    !*********************************************************
    ! Routine:  PrensaCtrlColoc()
    !*********************************************************
    FUNC bool PrensaCtrlColoc()
        VAR bool bPrnColocKo:=FALSE;

        IF DI_P240_PrnAuto=1 THEN
            USR_MsgWaitDI DI_P242_PrnOkColoc,s_AttesaDepoPrensa{nIdioma};
            WaitDI DI_P242_PrnOkColoc,1\MaxTime:=nTempoMaxDIPrnColoc\TimeFlag:=bPrnColocKo;
            IF bPrnColocKo=TRUE THEN
                Set DO_V08_LuzVermelha;
                ROB_AlarmeAcustico(2);
                USR_Print(s_CaricoPrensaKo{nIdioma});
                WaitTime nTempoMensAnom;
                Reset DO_V08_LuzVermelha;
                RETURN FALSE;
            ELSE
                RETURN TRUE;
            ENDIF
        ELSE
            Set DO_V08_LuzVermelha;
            ROB_AlarmeAcustico(2);
            USR_Print(s_AutomaticoPrensa{nIdioma});
            WaitTime nTempoMensAnom;
            Reset DO_V08_LuzVermelha;
            RETURN FALSE;
        ENDIF

    ENDFUNC

    !*********************************************************
    ! Routine:  PrensaCtrlPega()
    !*********************************************************
    FUNC bool PrensaCtrlPega()
        VAR bool bPrnPegalKo:=FALSE;

        IF DI_P240_PrnAuto=1 THEN
            USR_MsgWaitDI DI_P243_PrnOkPega,s_AttesaPrelievoPrensa{nIdioma};
            WaitDI DI_P243_PrnOkPega,1\MaxTime:=nTempoMaxDIPrnPega\TimeFlag:=bPrnPegalKo;
            IF bPrnPegalKo=TRUE THEN
                Set DO_V08_LuzVermelha;
                ROB_AlarmeAcustico(2);
                USR_Print(s_ErrPrelievoPrensa{nIdioma});
                WaitTime nTempoMensAnom;
                Reset DO_V08_LuzVermelha;
                RETURN FALSE;
            ELSE
                RETURN TRUE;
            ENDIF
        ELSE
            Set DO_V08_LuzVermelha;
            ROB_AlarmeAcustico(2);
            USR_Print(s_AutomaticoPrensa{nIdioma});
            WaitTime nTempoMensAnom;
            Reset DO_V08_LuzVermelha;
            RETURN FALSE;
        ENDIF

    ENDFUNC

    !*********************************************************
    ! Routine:  mENF_Cuba()
    !*********************************************************
    PROC mENF_Cuba()

        USR_Print(s_CicloRaffr{nIdioma});

        !MoveJ ENF_p01, vmax, z100, USR_toolGarra\WObj:=wobjMDF;
        !MoveJ ENF_p02, vmax, z100, USR_toolGarra\WObj:=wobjMDF;
        !MoveJ ENF_p03, vmax, z50, USR_toolGarra\WObj:=wobjMDF;
        !MoveJ ENF_p04, vmax, z50, USR_toolGarra\WObj:=wobjMDF;

        ! ===>>> POSICAO de Esfriamento <<<===
        !MoveL ENF_pCuba, v800, fine, USR_toolGarra\WObj:=wobjMDF;
        MoveJ ENF_pCuba,v150,fine,USR_toolGarra\WObj:=wobjMDF;
        ! ======================================
        USR_Print(s_AttesaRaff{nIdioma});
        WaitTime nTempoEsfriam;

        MoveL ENF_p01,v150,z50,USR_toolGarra\WObj:=wobjMDF;
        MoveJ ENF_p11,v150,z50,USR_toolGarra\WObj:=wobjMDF;
        ! MoveJ ENF_p12, v100, z50, USR_toolGarra\WObj:=wobjMDF;

        ! ===> POSICAO de GOTEJAMENTO <===
        MoveL ENF_p20,v80,fine,USR_toolGarra\WObj:=wobjMDF;
        MoveL ENF_p30,v80,fine,USR_toolGarra\WObj:=wobjMDF;
        ! =================================
        USR_Print(s_AttesaSgocc{nIdioma});
        WaitTime nTempoGotejamento;

        MoveJ ENF_p22,v600,z100,USR_toolGarra\WObj:=wobjMDF;
        !MoveJ ENF_p23, v600, z100, USR_toolGarra\WObj:=wobjMDF;

    ENDPROC

    !*********************************************************
    ! Routine:  mDEP_UtilIntColoc()
    !*********************************************************
    PROC mDEP_UtilIntColoc()

        USR_Print(s_UtilDepo{nIdioma});

        MoveJ UTL_p01,v2000,z100,USR_toolGarra\WObj:=wobjMDF;
        !MoveJ UTL_p02, v2000, z100, USR_toolGarra\WObj:=wobjMDF;
        !MoveJ UTL_p03, v2000, z100, USR_toolGarra\WObj:=wobjMDF;
        !MoveL UTL_p04, v2000, z50, USR_toolGarra\WObj:=wobjMDF;
        MoveL Offs(UTL_pColoc,0,0,400),v600,fine,USR_toolGarra\WObj:=wobjMDF;

        ! ===>>> POSICAO DE COLOCACAO <<<===
        MoveL UTL_pColoc,v30,fine,USR_toolGarra\WObj:=wobjMDF;
        ! =====================================
        ROB_GarraAbrir;
        nTipoPcNaPinca:=0;
        bPcColocada:=TRUE;

        MoveL Offs(UTL_pColoc,0,0,200),v800,fine,USR_toolGarra\WObj:=wobjMDF;
        MoveJ UTL_p11,vmax,z100,USR_toolGarra\WObj:=wobjMDF;
        !MoveJ UTL_p12, v1500, z100, USR_toolGarra\WObj:=wobjMDF;

        ! control sensor
        IF (bHbltcSnsUtilInt=TRUE AND DI_W17_SnsUtilIntermedio=0) THEN
            USR_Print(s_UtilSnsDeact{nIdioma});
            Set DO_V08_LuzVermelha;
            ROB_AlarmeAcustico(2);
            Reset DO_P006_AnomaliaRobo;
            PulseDO\PLength:=2,DO_P006_AnomaliaRobo;
            USR_Print(s_AttesaReset{nIdioma});
            WaitDI DI_V01_ResetAllRob,1;
            Reset DO_V08_LuzVermelha;
        ENDIF

    ENDPROC

    !*********************************************************
    ! Routine:  mDEP_UtilIntRecoc()
    !*********************************************************
    PROC mDEP_UtilIntPega()

        USR_Print(s_UtilPrel{nIdioma});

        MoveJ UTL_p51,v5000,z100,USR_toolGarra\WObj:=wobjMDF;
        !MoveJ UTL_p52, vmax, z100, USR_toolGarra\WObj:=wobjMDF;
        !MoveJ UTL_p53, vmax, z100, USR_toolGarra\WObj:=wobjMDF;
        !MoveL UTL_p54, v1500, z50, USR_toolGarra\WObj:=wobjMDF;
        MoveL Offs(UTL_pPega,0,0,200),v800,fine,USR_toolGarra\WObj:=wobjMDF;

        ! ===>>> POSICAO DE RETIRADA <<<===
        MoveL UTL_pPega,v100,fine,USR_toolGarra\WObj:=wobjMDF;
        ! ==================================
        ROB_GarraFechar;
        nTipoPcNaPinca:=1;
        bPcColocada:=FALSE;

        MoveL Offs(UTL_pPega,0,0,200),v1000,fine,USR_toolGarra\WObj:=wobjMDF;
        !MoveJ UTL_p61, vmax, z100, USR_toolGarra\WObj:=wobjMDF;
        MoveJ UTL_p62,v1500,z100,USR_toolGarra\WObj:=wobjMDF;
        MoveJ UTL_p82,v1500,z100,USR_toolGarra\WObj:=wobjMDF;
        !MoveJ UTL_p72, vmax, z100, USR_toolGarra\WObj:=wobjMDF;

        ! control sensor
        IF (bHbltcSnsUtilInt=TRUE AND DI_W17_SnsUtilIntermedio=1) THEN
            USR_Print(s_UtilSnsAct{nIdioma});
            Set DO_W02_LuzAmarelo;
            ROB_AlarmeAcustico(2);
            Reset DO_P006_AnomaliaRobo;
            PulseDO\PLength:=2,DO_P006_AnomaliaRobo;
            WaitTime nTempoMensAnom;
            Reset DO_W02_LuzAmarelo;
        ENDIF

    ENDPROC

    !*********************************************************
    ! Routine:  mDEP_PrnColoc()
    !*********************************************************
    PROC mDEP_PrnColoc()

        USR_Print(s_DepositoPrensa{nIdioma});

        MoveJ PRN_p01,v2500,z100,USR_toolGarra\WObj:=wobjMDF;
        !
        ! Quebra de Rebarba...
        MoveJ pQuebraRebarba_00,v1500,z30,USR_toolGarra\WObj:=wobjMDF;
        MoveJ pQuebraRebarba_01,v800,z30,USR_toolGarra\WObj:=wobjMDF;
        MoveJ pQuebraRebarba_02,v600,z30,USR_toolGarra\WObj:=wobjMDF;
        MoveJ pQuebraRebarba_02,v1000,z30,USR_toolGarra\WObj:=wobjMDF;
        MoveJ pQuebraRebarba_00,v1500,z30,USR_toolGarra\WObj:=wobjMDF;
        !
        MoveJ PRN_p01,v2500,z100,USR_toolGarra\WObj:=wobjMDF;

        ! ===>>> POSICAO FUERA de la PRENSA!!! <<<===
        MoveJDO PRN_p02,v800,z100,USR_toolGarra\WObj:=wobjMDF,DO_V06_PrensaForaAreaTrab_User,0;
        ! ============================================

        MoveJ PRN_p03,v1000,z100,USR_toolGarra\WObj:=wobjMDF;
        !MoveL PRN_p04, v1000, z100, USR_toolGarra\WObj:=wobjMDF;
        !MoveJ PRN_p05, v800, z50, USR_toolGarra\WObj:=wobjMDF;
        !
        !    Defino a posicao de deposito como sendo uma para cada retirada da gaveta
        !
        TEST nRetirouDaGaveta
            CASE 1:
                PRN_pColoc := pDepositaPrensa_1;
            CASE 2:
                PRN_pColoc := pDepositaPrensa_2;
            CASE 3:
                PRN_pColoc := pDepositaPrensa_3;
            CASE 4:
                PRN_pColoc := pDepositaPrensa_4;
            CASE 5:
                PRN_pColoc := pDepositaPrensa_5;
            CASE 6:
                PRN_pColoc := pDepositaPrensa_6;
            DEFAULT:
                PRN_pColoc := PRN_pColoc;
                Stop;
        ENDTEST


        !
        !
        !pDepositaPrensa_1 := PRN_pColoc;
        !
        MoveJ Offs(PRN_pColoc,0,0,250),v400,fine,USR_toolGarra\WObj:=wobjMDF;

        ! ===>>> POSICAO de COLOCACAO <<<===
        MoveL PRN_pColoc,v200,fine,USR_toolGarra\WObj:=wobjMDF;
        ! ====================================

        ROB_GarraAbrir;
        nTipoPcNaPinca:=0;
        bPcColocada:=TRUE;

        !MoveL PRN_p10, v500, z10, USR_toolGarra\WObj:=wobjMDF;
        MoveL Offs(PRN_pColoc,0,0,200),v600,fine,USR_toolGarra\WObj:=wobjMDF;
        MoveL PRN_p11,v1000,z50,USR_toolGarra\WObj:=wobjMDF;
        !MoveJ PRN_p12, vmax, z100, USR_toolGarra\WObj:=wobjMDF;

        ! ===>>> POSICAO FUERA de la PRENSA!!! <<<===
        MoveJDO PRN_p13,v800,z5,USR_toolGarra\WObj:=wobjMDF,DO_V06_PrensaForaAreaTrab_User,1;
        ! ============================================

        MoveJ PRN_p14,vmax,fine,USR_toolGarra\WObj:=wobjMDF;

        USR_Print(s_StartPrensa{nIdioma});
        WaitTime\inpos,0;
        Reset DO_P242_PrnStartAposColoc;
        PulseDO\PLength:=1,DO_P242_PrnStartAposColoc;

        Reset DO_P033_PcColocPrensa;
        PulseDO\PLength:=1,DO_P033_PcColocPrensa;

        WaitDI DI_P242_PrnOkColoc,0\MaxTime:=1\TimeFlag:=bPrnErrStart1;
        IF bPrnErrStart1=TRUE THEN
            ROB_AlarmeAcustico(2);
            USR_Print(s_PrensaNonPartita{nIdioma});
            WaitTime nTempoMensAnom;
        ENDIF

    ENDPROC

    !*********************************************************
    ! Routine:  mDEP_PrnPega()
    !*********************************************************
    PROC mDEP_PrnPega()

        USR_Print(s_PrelievoPrensa{nIdioma});
        Set DO_W09_AbrirGarra;
        nTipoPcNaPinca:=0;
        bPcColocada:=TRUE;

        MoveJ PRN_p50,vmax,z100,USR_toolGarra\WObj:=wobjMDF;

        ! ===>>> POSICAO FUERA de la PRENSA!!! <<<===
        MoveJDO PRN_p51,vmax,z50,USR_toolGarra\WObj:=wobjMDF,DO_V06_PrensaForaAreaTrab_User,0;
        ! ============================================

        MoveJ PRN_p52,vmax,z100,USR_toolGarra\WObj:=wobjMDF;
        MoveJ PRN_p53,vmax,z100,USR_toolGarra\WObj:=wobjMDF;
        MoveL PRN_p54,vmax,z10,USR_toolGarra\WObj:=wobjMDF;

        ! ===>>> POSICAO de RETIRADA <<<===
        MoveL PRN_pPega,v300,fine,USR_toolGarra\WObj:=wobjMDF;
        ! ==================================

        IF bHbltcPrnPegaSoft=TRUE THEN
            SoftAct 1,100;
            ! SoftAct 2,10;
            ! SoftAct 3,10;
            SoftAct 4,10;
            SoftAct 5,10;
            SoftAct 6,10;
            WaitTime nTempoGarraFechar;
            !Tempo espera pasaje hacia ejes soft
        ENDIF

        ROB_GarraFechar;
        nTipoPcNaPinca:=1;
        bPcColocada:=FALSE;

        IF bHbltcPrnPegaSoft=TRUE THEN
            WaitTime 1;
            WaitTime\inpos,0;
            PRN_pTemp:=CRobT(\Tool:=USR_toolGarra\WObj:=wobjMDF);
            SoftDeact;
            MoveL Offs(PRN_pTemp,0,0,300),v100,fine,USR_toolGarra\WObj:=wobjMDF;
            WaitTime\inpos,0;
            SoftDeact;
        ENDIF

        MoveL PRN_p60,v1500,fine,USR_toolGarra\WObj:=wobjMDF;
        MoveL PRN_p61,vmax,fine,USR_toolGarra\WObj:=wobjMDF;
        MoveL PRN_p62,vmax,z100,USR_toolGarra\WObj:=wobjMDF;

        ! ===>>> POSICAO FUERA de la PRENSA!!! <<<===
        MoveJDO PRN_p63,vmax,z5,USR_toolGarra\WObj:=wobjMDF,DO_V06_PrensaForaAreaTrab_User,1;
        ! ============================================

        MoveJ PRN_p64,vmax,z100,USR_toolGarra\WObj:=wobjMDF;

        USR_Print(s_StartPrensa{nIdioma});
        WaitTime\inpos,0;
        Reset DO_P243_PrnStartAposPega;
        PulseDO\PLength:=1,DO_P243_PrnStartAposPega;

        Reset DO_P044_PcPegaPrensa;
        PulseDO\PLength:=1,DO_P044_PcPegaPrensa;

        WaitDI DI_P243_PrnOkPega,0\MaxTime:=1\TimeFlag:=bPrnErrStart2;
        IF bPrnErrStart2=TRUE THEN
            ROB_AlarmeAcustico(2);
            USR_Print(s_PrensaNonPartita{nIdioma});
            WaitTime nTempoMensAnom;
        ENDIF

    ENDPROC

    PROC PresaSoft()

        ROB_GarraAbrir;
        MoveL p01,v500,fine,USR_toolGarra\WObj:=wobjMDF;
        MoveL p02,v300,fine,USR_toolGarra\WObj:=wobjMDF;

        SoftAct 1,100;
        ! SoftAct 2,10;
        ! SoftAct 3,10;
        SoftAct 4,10;
        SoftAct 5,10;
        SoftAct 6,10;
        WaitTime nTempoGarraFechar;

        ROB_GarraFechar;

        WaitTime 1;
        WaitTime\inpos,0;
        pTemp:=CRobT(\Tool:=USR_toolGarra\WObj:=wobjMDF);
        MoveL Offs(pTemp,0,0,200),v300,fine,USR_toolGarra\WObj:=wobjMDF;
        WaitTime\inpos,0;
        SoftDeact;

        MoveL p01,v500,fine,USR_toolGarra\WObj:=wobjMDF;

    ENDPROC

    !*********************************************************
    ! Routine:  mDEP_PcPrensadaColoc()
    !*********************************************************
    PROC mDEP_PcPrensadaColoc()

        USR_Print(s_DepositoPrensati{nIdioma});

        MoveJ PRD_p01,vmax,z100,USR_toolGarra\WObj:=wobjMDF;
        MoveJ PRD_p02,vmax,z100,USR_toolGarra\WObj:=wobjMDF;
        MoveJ PRD_p03,vmax,z100,USR_toolGarra\WObj:=wobjMDF;
        MoveJ PRD_p04,v600,z20,USR_toolGarra\WObj:=wobjMDF;
        MoveL PRD_p05,v400,fine,USR_toolGarra\WObj:=wobjMDF;

        ! ===>>> POSICAO de COLOCACAO <<<===
        MoveL PRD_pColoc,v300,fine,USR_toolGarra\WObj:=wobjMDF;
        ! ====================================

        ROB_GarraAbrir;
        MoveL Offs(PRD_pColoc,0,0,120),v300,fine,USR_toolGarra\WObj:=wobjMDF;
        nTipoPcNaPinca:=0;
        bPcColocada:=TRUE;

        MoveL PRD_p10,v500,z50,USR_toolGarra\WObj:=wobjMDF;
        MoveL PRD_p11,vmax,z100,USR_toolGarra\WObj:=wobjMDF;
        MoveJ PRD_p12,vmax,z100,USR_toolGarra\WObj:=wobjMDF;
        MoveJ PRD_p13,vmax,z100,USR_toolGarra\WObj:=wobjMDF;
        MoveJ PRD_p14,vmax,z100,USR_toolGarra\WObj:=wobjMDF;

        Reset DO_P035_PcColocEsteiraRejeicao;
        PulseDO\PLength:=nTempPulsoEsteira,DO_P034_PcColocEsteiraBoa;

    ENDPROC

    !*********************************************************
    ! Routine:  mDEP_PcBoaColoc()
    !*********************************************************
    PROC mDEP_PcBoaColoc()

        IF bQualidade=TRUE THEN
            ROB_AlarmeAcustico(2);
            USR_Print(s_DepQualita{nIdioma});
        ELSE
            USR_Print(s_DepositoBuono{nIdioma});
        ENDIF

        MoveJ BUE_p01,vmax,z100,USR_toolGarra\WObj:=wobjMDF;
        MoveJ BUE_p02,vmax,z100,USR_toolGarra\WObj:=wobjMDF;
        MoveJ BUE_p03,vmax,z100,USR_toolGarra\WObj:=wobjMDF;
        MoveL BUE_p04,vmax,z100,USR_toolGarra\WObj:=wobjMDF;
        MoveL BUE_p05,v800,z50,USR_toolGarra\WObj:=wobjMDF;

        ! ===>>> POSICAO de COLOCACAO <<<===
        MoveL BUE_pColoc,v500,fine,USR_toolGarra\WObj:=wobjMDF;
        ! ====================================

        ROB_GarraAbrir;
        nTipoPcNaPinca:=0;
        bPcColocada:=TRUE;
        IF bQualidade=TRUE THEN
            bQualidade:=FALSE;
            Reset DO_W02_LuzAmarelo;
        ENDIF

        MoveL BUE_p10,v800,z50,USR_toolGarra\WObj:=wobjMDF;
        MoveL BUE_p11,vmax,z100,USR_toolGarra\WObj:=wobjMDF;
        MoveJ BUE_p12,vmax,z100,USR_toolGarra\WObj:=wobjMDF;
        MoveJ BUE_p13,vmax,z100,USR_toolGarra\WObj:=wobjMDF;
        !MoveJ BUE_p14, vmax, z100, USR_toolGarra\WObj:=wobjMDF;

        Reset DO_P034_PcColocEsteiraBoa;
        PulseDO\PLength:=1,DO_P034_PcColocEsteiraBoa;

    ENDPROC

    !*********************************************************
    ! Routine:  mDEP_PcRejeicaoColoc()
    !*********************************************************
    PROC mDEP_PcRejeicaoColoc()

        USR_Print(s_DepositoScarto{nIdioma});

        MoveJ RCZ_p01,vmax,z100,USR_toolGarra\WObj:=wobjMDF;
        MoveJ RCZ_p02,vmax,z100,USR_toolGarra\WObj:=wobjMDF;
        !MoveJ RCZ_p03, vmax, z100, USR_toolGarra\WObj:=wobjMDF;
        !MoveL RCZ_p04, vmax, z100, USR_toolGarra\WObj:=wobjMDF;
        !MoveJ RCZ_p05, v500, z50, USR_toolGarra\WObj:=wobjMDF;

        ! ===>>> POSICAO de COLOCACAO <<<===
        MoveL RCZ_pColoc,v300,fine,USR_toolGarra\WObj:=wobjMDF;
        ! ====================================

        ROB_GarraAbrir;
        nTipoPcNaPinca:=0;
        bPcColocada:=TRUE;

        MoveL RCZ_p10,v500,z50,USR_toolGarra\WObj:=wobjMDF;
        MoveJ RCZ_p11,vmax,z100,USR_toolGarra\WObj:=wobjMDF;
        MoveJ RCZ_p12,vmax,z100,USR_toolGarra\WObj:=wobjMDF;
        MoveJ RCZ_p13,vmax,z100,USR_toolGarra\WObj:=wobjMDF;
        !MoveL RCZ_p14, vmax, z100, USR_toolGarra\WObj:=wobjMDF;
        MoveJ RCZ_p14,vmax,z100,USR_toolGarra\WObj:=wobjMDF;

        Reset DO_P035_PcColocEsteiraRejeicao;
        PulseDO\PLength:=1,DO_P035_PcColocEsteiraRejeicao;

    ENDPROC

    !*********************************************************
    ! Routine:  MDF_AnomaliaExtracao()
    !*********************************************************
    PROC MDF_AnomaliaExtracao()
        VAR bool bVerifInyecc:=FALSE;

        IF bInjecaoKo=TRUE THEN
            USR_Print(s_EstrazioneFallita{nIdioma});
        ELSEIF bMassaloteKo=TRUE THEN
            USR_Print(s_MaterozzaNonOk{nIdioma});
        ENDIF

        WaitTime\inpos,0;
        SpeedRefresh 100;

        Set DO_V08_LuzVermelha;
        ROB_AlarmeAcustico(2);
        Reset DO_P015_PcIncompleta;
        PulseDO\PLength:=2,DO_P015_PcIncompleta;
        Reset DO_P006_AnomaliaRobo;
        PulseDO\PLength:=2,DO_P006_AnomaliaRobo;

        USR_Print(s_AttesaReset{nIdioma});
        WHILE DI_V01_ResetAllRob=0 DO
            IF DI_P002_InjecaoOk=0 bVerifInyecc:=TRUE;
            WaitTime 0.1;
        ENDWHILE
        Reset DO_V08_LuzVermelha;
        Reset DO_P015_PcIncompleta;

        IF bVerifInyecc=FALSE THEN
            IF (nHbltcMensajes=1 OR (nHbltcMensajes=2 AND DOutput(DO_V07_RobEmAuto)=1)) THEN
                USR_Print(s_AttesaIniezOkReset{nIdioma});
            ENDIF
            WaitDI DI_P002_InjecaoOk,0;
        ENDIF

    ENDPROC

    !*********************************************************
    ! Routine:  zROB_PosTransporte()
    !*********************************************************
    PROC zROB_PosTransporte()

        MoveAbsJ jposTransporte\NoEOffs,v1000,fine,tool0;

    ENDPROC


    !*********************************************************
    ! Routine:  zROB_PosCalibracao()
    !*********************************************************
    PROC zROB_PosCalibracao()

        MoveAbsJ jposCalib\NoEOffs,v1000,fine,tool0;

    ENDPROC


    !*********************************************************
    ! Routine:  zROB_PosMontaStampi()
    !*********************************************************
    PROC zROB_PosMontaStampi()

        MoveJ ROB_pHome,v1000,z5,USR_toolGarra\WObj:=wobjMDF;
        MoveJ MMD_p01,v1000,z5,USR_toolGarra\WObj:=wobjMDF;
        MoveJ MMD_p02,v1000,fine,USR_toolGarra\WObj:=wobjMDF;
        Stop;
        MoveJ MMD_p01,v1000,z5,USR_toolGarra\WObj:=wobjMDF;
        MoveJ ROB_pHome,v1000,z5,USR_toolGarra\WObj:=wobjMDF;

    ENDPROC

    !*********************************************************
    ! Routine:  zTeach_Positions()
    ! Advertencia: lista de todas las posiciones. Esta rutina no
    !              es llamada de la rotina Main(), ma es solamente
    !              un resumen para simplificar la memorizacion
    !              de las posiciones.
    ! IMPORTANTE: Si desea a?adir y/o eliminar una POSICAO que
    !             tiene que hacer en la misma rutina, no s?lo aqu?!!
    !             Incluso VELOCIDAD 'y aproximaCAO deber?a ser
    !             modificados en la misma rutina.
    !*********************************************************
    PROC zTeach_Positions()

        ! IMPORTANTE: DEBE SER POSIBLE PASAR DE LA ?LTIMA POSICAO
        ! DE CUALQUIER "mRUTINA" A LA POSICAO INICIAL SIN COLISIONES!!!

        ! >>> mROB_Home: POSICAO inicial (home position)
        MoveJ ROB_pHome,vmax,z5,USR_toolGarra\wobj:=wobjMDF;

        ! >>> mMDF_Espera: POSICAO de espera en frente de la puerta de la m?quina
        MoveL MDF_pEspera,vmax,z5,USR_toolGarra\wobj:=wobjMDF;

        ! >>> mMDF_Pega: entrada en m?quina y pega de la PECA
        ! en linea con el centro del molde, sobre la columna baja
        MoveJ MDF_p01,vmax,z50,USR_toolGarra\WObj:=wobjMDF;
        ! centro del molde, en linea con la massalote
        MoveJ MDF_p02,vmax,z50,USR_toolGarra\WObj:=wobjMDF;
        ! en linea con la massalote, levemente antes
        MoveL MDF_p03,v3000,z50,USR_toolGarra\WObj:=wobjMDF;
        ! ===>>> POSICAO de RETIRADA <<<===
        MoveL MDF_pPega,v300,fine,USR_toolGarra\WObj:=wobjMDF;
        ! en linea con la massalote, levemente m?s all? de la carrera
        ! m?xima de la eyecCAO
        MoveL MDF_p04,v1000,fine,USR_toolGarra\WObj:=wobjMDF;

        ! >>> mMDF_Saida: salida de la m?quina hasta fuera ?rea
        ! centro del molde, en linea con la massalote
        MoveL\Conc,MDF_p10,v3000,z30,USR_toolGarra\WObj:=wobjMDF;
        ! en linea con el centro del molde, acerca de la columna
        MoveL\Conc,MDF_p11,vmax,z50,USR_toolGarra\wobj:=wobjMDF;
        ! POSICAO hasta la salida de la m?quina
        MoveJ MDF_p12,vmax,z50,USR_toolGarra\wobj:=wobjMDF;
        ! posiciones acercando sensor start pulverizador (si presente...)
        !MoveJ MDF_p20, vmax, z50, USR_toolGarra\WObj:=wobjMDF;
        !MoveJ MDF_p21, v2000, z50, USR_toolGarra\WObj:=wobjMDF;
        ! ===>>> POSICAO de CONTROL START PULVER. <<<=== (si presente...)
        MoveL MDF_pControl,v1000,fine,USR_toolGarra\WObj:=wobjMDF;
        ! posiciones que se alejan del sensor (si presente...)
        MoveJ MDF_p30,v2000,z50,USR_toolGarra\WObj:=wobjMDF;
        MoveJ MDF_p31,vmax,z50,USR_toolGarra\WObj:=wobjMDF;
        ! POSICAO hasta salida de la m?quin
        MoveJ MDF_p13,vmax,z50,USR_toolGarra\WObj:=wobjMDF;
        ! ===>>> POSICAO FUERA de la PUERTA de la M?QUINA!!! <<<===
        MoveJ MDF_p14,vmax,z50,USR_toolGarra\WObj:=wobjMDF;

        ! >>> mSNS_ControlPc: sensores
        ! posiciones acercando
        MoveJ SNS_p01,vmax,z100,USR_toolGarra\WObj:=wobjMDF;
        MoveJ SNS_p02,v2000,z50,USR_toolGarra\WObj:=wobjMDF;
        ! ===>>> 1a POSICAO de CONTROL <<<===
        MoveL SNS_pControl1,v500,fine,USR_toolGarra\WObj:=wobjMDF;
        ! ===>>> 2a POSICAO de CONTROL <<<===
        MoveL SNS_pControl2,v500,fine,USR_toolGarra\WObj:=wobjMDF;
        ! ===>>> 3a POSICAO de CONTROL <<<===
        MoveL SNS_pControl3,v500,fine,USR_toolGarra\WObj:=wobjMDF;
        ! ===>>> 4a POSICAO de CONTROL <<<===
        MoveL SNS_pControl4,v500,fine,USR_toolGarra\WObj:=wobjMDF;
        ! posiciones que se alejan
        MoveJ SNS_p10,v2000,z50,USR_toolGarra\WObj:=wobjMDF;
        MoveJ SNS_p11,vmax,z100,USR_toolGarra\WObj:=wobjMDF;

        ! >>> mENF_Cuba: Esfriamento en la cuba de agua
        ! posiciones acercando
        !MoveJ ENF_p01, vmax, z100, USR_toolGarra\WObj:=wobjMDF;
        !MoveJ ENF_p02, vmax, z100, USR_toolGarra\WObj:=wobjMDF;
        !MoveJ ENF_p03, v1000, z50, USR_toolGarra\WObj:=wobjMDF;
        !MoveJ ENF_p04, v1000, z50, USR_toolGarra\WObj:=wobjMDF;
        ! ===>>> POSICAO de Esfriamento <<<===
        MoveL ENF_pCuba,v300,fine,USR_toolGarra\wobj:=wobjMDF;
        ! posiciones hasta gotejamento
        MoveJ ENF_p10,v100,z50,USR_toolGarra\WObj:=wobjMDF;
        !MoveJ ENF_p11, v100, z50, USR_toolGarra\WObj:=wobjMDF;
        !MoveJ ENF_p12, v100, z50, USR_toolGarra\WObj:=wobjMDF;
        ! ===> POSICAO de GOTEJAMENTO <===
        MoveL ENF_p20,v100,fine,USR_toolGarra\WObj:=wobjMDF;
        ! posiciones que se alejan
        MoveJ ENF_p21,v1000,z50,USR_toolGarra\WObj:=wobjMDF;
        MoveJ ENF_p22,v2000,z1,USR_toolGarra\WObj:=wobjMDF;
        !MoveJ ENF_p23, vmax, z100, USR_toolGarra\WObj:=wobjMDF;

        ! >>> mDEP_UtilIntColoc: colocaCAO PECA en util intermedio
        ! posiciones acercando
        MoveJ UTL_p01,vmax,z100,USR_toolGarra\WObj:=wobjMDF;
        !MoveJ UTL_p02, vmax, z100, USR_toolGarra\WObj:=wobjMDF;
        !MoveJ UTL_p03, v1500, z50, USR_toolGarra\WObj:=wobjMDF;
        MoveL UTL_p04,v200,fine,USR_toolGarra\WObj:=wobjMDF;
        ! ===>>> POSICAO DE COLOCACAO <<<===
        MoveL Offs(UTL_pColoc,0,0,200),v200,fine,USR_toolGarra\WObj:=wobjMDF;
        MoveL UTL_pColoc,v200,fine,USR_toolGarra\WObj:=wobjMDF;
        ! posiciones que se alejan
        MoveL Offs(UTL_pColoc,0,0,200),v200,fine,USR_toolGarra\WObj:=wobjMDF;
        !MoveL UTL_p10, v800, z50, USR_toolGarra\WObj:=wobjMDF;
        !MoveJ UTL_p11, v1500, z50, USR_toolGarra\WObj:=wobjMDF;
        !MoveJ UTL_p12, v1500, z50, USR_toolGarra\WObj:=wobjMDF;

        ! >>> mDEP_UtilIntRecoc: pega PECA de util intermedio
        ! posiciones acercando
        !MoveJ UTL_p51, vmax, z100, USR_toolGarra\WObj:=wobjMDF;
        !MoveJ UTL_p52, vmax, z100, USR_toolGarra\WObj:=wobjMDF;
        !MoveJ UTL_p53, v1500, z50, USR_toolGarra\WObj:=wobjMDF;
        !MoveL UTL_p54, v400, fine, USR_toolGarra\WObj:=wobjMDF;
        MoveL Offs(UTL_pPega,0,0,200),v200,fine,USR_toolGarra\WObj:=wobjMDF;
        ! ===>>> POSICAO DE RETIRADA <<<===
        MoveL UTL_pPega,v200,fine,USR_toolGarra\WObj:=wobjMDF;
        ! posiciones que se alejan
        MoveL UTL_p60,v800,z50,USR_toolGarra\WObj:=wobjMDF;
        !MoveJ UTL_p61, v1500, z50, USR_toolGarra\WObj:=wobjMDF;
        !MoveJ UTL_p62, v1500, z50, USR_toolGarra\WObj:=wobjMDF;

        ! >>> mDEP_PrnColoc: colocaCAO PECA en la prensa
        ! POSICAO acercando
        MoveJ PRN_p01,vmax,z100,USR_toolGarra\WObj:=wobjMDF;
        ! === POSICAO FUERA de la PRENSA!!! ===
        !MoveJDO PRN_p02, vmax, z100, USR_toolGarra\WObj:=wobjMDF, DO_V06_PrensaForaAreaTrab_User, 0;
        ! posiciones acercando
        MoveJ PRN_p03,v1500,z50,USR_toolGarra\WObj:=wobjMDF;
        !MoveL PRN_p04, v1500, z50, USR_toolGarra\WObj:=wobjMDF;
        !MoveL PRN_p05, v1500, z50, USR_toolGarra\WObj:=wobjMDF;
        MoveL Offs(PRN_pColoc,0,0,200),v500,fine,USR_toolGarra\WObj:=wobjMDF;
        ! ===>>> POSICAO de COLOCACAO <<<===
        MoveL PRN_pColoc,v100,fine,USR_toolGarra\WObj:=wobjMDF;
        ! posiciones que se alejan
        MoveL PRN_p10,v500,z1,USR_toolGarra\WObj:=wobjMDF;
        MoveL PRN_p11,v500,z10,USR_toolGarra\WObj:=wobjMDF;
        MoveL PRN_p12,v1500,z50,USR_toolGarra\WObj:=wobjMDF;
        ! === POSICAO FUERA de la PRENSA!!! ===
        MoveJ PRN_p13,vmax,z5,USR_toolGarra\WObj:=wobjMDF;
        ! posiciones que se alejan
        MoveJ PRN_p14,vmax,z50,USR_toolGarra\WObj:=wobjMDF;

        ! >>> mDEP_PrnPega: pega PECA en la prensa
        ! POSICAO acercando
        MoveJ PRN_p50,vmax,z100,USR_toolGarra\WObj:=wobjMDF;
        ! === POSICAO FUERA de la PRENSA!!! ===
        MoveJDO PRN_p51,vmax,z50,USR_toolGarra\WObj:=wobjMDF,DO_V06_PrensaForaAreaTrab_User,0;
        ! posiciones acercando
        MoveJ PRN_p52,v1500,z50,USR_toolGarra\WObj:=wobjMDF;
        MoveL PRN_p53,v1000,z50,USR_toolGarra\WObj:=wobjMDF;
        MoveL PRN_p54,v500,z10,USR_toolGarra\WObj:=wobjMDF;
        ! ===>>> POSICAO de RETIRADA <<<===
        MoveL PRN_pPega,v300,fine,USR_toolGarra\WObj:=wobjMDF;
        ! posiciones que se alejan
        MoveL PRN_p60,v300,z1,USR_toolGarra\WObj:=wobjMDF;
        MoveL PRN_p61,v1000,z10,USR_toolGarra\WObj:=wobjMDF;
        MoveL PRN_p62,v1500,z50,USR_toolGarra\WObj:=wobjMDF;
        ! === POSICAO FUERA de la PRENSA!!! ===
        MoveJ PRN_p63,vmax,z5,USR_toolGarra\WObj:=wobjMDF;
        ! posiciones que se alejan
        MoveJ PRN_p64,vmax,z50,USR_toolGarra\WObj:=wobjMDF;

        ! >>> mDEP_PcPrensadaColoc: colocaCAO PECA prensada
        ! posiciones acercando
        MoveJ PRD_p01,vmax,z100,USR_toolGarra\WObj:=wobjMDF;
        MoveJ PRD_p02,vmax,z100,USR_toolGarra\WObj:=wobjMDF;
        MoveJ PRD_p03,v1500,z50,USR_toolGarra\WObj:=wobjMDF;
        MoveL PRD_p04,v1500,z50,USR_toolGarra\WObj:=wobjMDF;
        MoveL PRD_p05,v500,z50,USR_toolGarra\WObj:=wobjMDF;
        ! ===>>> POSICAO de COLOCACAO <<<===
        MoveL PRD_pColoc,v300,fine,USR_toolGarra\WObj:=wobjMDF;
        ! posiciones que se alejan
        MoveL PRD_p10,v500,z50,USR_toolGarra\WObj:=wobjMDF;
        MoveL PRD_p11,v1000,z50,USR_toolGarra\WObj:=wobjMDF;
        MoveJ PRD_p12,v1500,z50,USR_toolGarra\WObj:=wobjMDF;
        MoveJ PRD_p13,vmax,z100,USR_toolGarra\WObj:=wobjMDF;
        MoveJ PRD_p14,vmax,z100,USR_toolGarra\WObj:=wobjMDF;

        ! >>> mDEP_PcBoaColoc: deposito pezzi buoni/qualit?
        ! posiciones acercando
        MoveJ BUE_p01,vmax,z100,USR_toolGarra\WObj:=wobjMDF;
        MoveJ BUE_p02,vmax,z100,USR_toolGarra\WObj:=wobjMDF;
        MoveJ BUE_p03,v1500,z50,USR_toolGarra\WObj:=wobjMDF;
        MoveL BUE_p04,v1500,z50,USR_toolGarra\WObj:=wobjMDF;
        MoveL BUE_p05,v500,z50,USR_toolGarra\WObj:=wobjMDF;
        ! ===>>> POSICAO de COLOCACAO <<<===
        MoveL BUE_pColoc,v300,fine,USR_toolGarra\WObj:=wobjMDF;
        ! posiciones que se alejan
        MoveL BUE_p10,v500,z50,USR_toolGarra\WObj:=wobjMDF;
        MoveL BUE_p11,v1000,z50,USR_toolGarra\WObj:=wobjMDF;
        MoveJ BUE_p12,v1500,z50,USR_toolGarra\WObj:=wobjMDF;
        MoveJ BUE_p13,vmax,z100,USR_toolGarra\WObj:=wobjMDF;
        MoveJ BUE_p14,vmax,z100,USR_toolGarra\WObj:=wobjMDF;

        ! >>> mDEP_PcRejeicaoColoc: deposito pezzi scarto
        ! posiciones acercando
        MoveJ RCZ_p01,vmax,z100,USR_toolGarra\WObj:=wobjMDF;
        MoveJ RCZ_p02,vmax,z100,USR_toolGarra\WObj:=wobjMDF;
        MoveJ RCZ_p03,v1500,z50,USR_toolGarra\WObj:=wobjMDF;
        MoveL RCZ_p04,v1500,z50,USR_toolGarra\WObj:=wobjMDF;
        MoveJ RCZ_p05,v500,z50,USR_toolGarra\WObj:=wobjMDF;
        ! ===>>> POSICAO de COLOCACAO <<<===
        MoveL RCZ_pColoc,v300,fine,USR_toolGarra\WObj:=wobjMDF;
        ! posiciones que se alejan
        MoveL RCZ_p10,v500,z50,USR_toolGarra\WObj:=wobjMDF;
        MoveL RCZ_p11,v1000,z50,USR_toolGarra\WObj:=wobjMDF;
        MoveJ RCZ_p12,v1500,z50,USR_toolGarra\WObj:=wobjMDF;
        MoveJ RCZ_p13,vmax,z100,USR_toolGarra\WObj:=wobjMDF;
        MoveJ RCZ_p14,vmax,z10,USR_toolGarra\WObj:=wobjMDF;

    ENDPROC

    PROC alcance()
        MoveJ [[-732.10,-870.12,2627.26],[0.782964,0.621049,0.0245496,-0.025745],[-1,-2,2,1],[9E+09,9E+09,9E+09,9E+09,9E+09,9E+09]],v1000,z50,USR_toolGarra\WObj:=wobjMDF;
        MoveJ [[-706.49,-1045.02,3027.08],[0.00369331,0.0070574,-0.621494,0.783378],[-1,-2,0,1],[9E+09,9E+09,9E+09,9E+09,9E+09,9E+09]],v1000,z50,USR_toolGarra\WObj:=wobjMDF;
        MoveL [[-706.49,-1482.04,3027.08],[0.00369225,0.00705501,-0.621493,0.783379],[0,-2,0,1],[9E+09,9E+09,9E+09,9E+09,9E+09,9E+09]],v1000,z50,USR_toolGarra\WObj:=wobjMDF;
        MoveJ [[-706.49,-1045.00,3027.08],[0.00369145,0.00705366,-0.621493,0.783379],[-1,-2,0,1],[9E+09,9E+09,9E+09,9E+09,9E+09,9E+09]],v1000,z50,USR_toolGarra\WObj:=wobjMDF;
        MoveJ [[-734.75,-1048.08,2817.04],[0.782842,0.620934,0.0273064,-0.0292195],[-1,-2,2,1],[9E+09,9E+09,9E+09,9E+09,9E+09,9E+09]],v1000,z50,USR_toolGarra\WObj:=wobjMDF;
        MoveL [[-734.75,-1487.10,2817.04],[0.782842,0.620934,0.0273071,-0.0292209],[0,-2,2,1],[9E+09,9E+09,9E+09,9E+09,9E+09,9E+09]],v1000,z50,USR_toolGarra\WObj:=wobjMDF;
    ENDPROC

    PROC mDepGaveta_1()
        MoveJ pDepGaveta_1_1,v1000,z50,USR_toolGarra\WObj:=wobjMDF;
        MoveJ pDepGaveta_1_11,v1000,z50,USR_toolGarra\WObj:=wobjMDF;
        !
        MoveJ pDepGaveta_1_21,v1000,z50,USR_toolGarra\WObj:=wobjMDF;
        MoveL pDepGaveta_1_31,v1000,z50,USR_toolGarra\WObj:=wobjMDF;
        MoveL pDepGaveta_1_41,v1000,z50,USR_toolGarra\WObj:=wobjMDF;
        MoveL pDepGaveta_1_51,v1000,z50,USR_toolGarra\WObj:=wobjMDF;
        MoveL pDepGaveta_1_61,v1000,z50,USR_toolGarra\WObj:=wobjMDF;
        MoveL pDepGaveta_1_71,v1000,z50,USR_toolGarra\WObj:=wobjMDF;
        !
        ROB_GarraAbrir;
        !
        MoveL pDepGaveta_1_81,v1000,z50,USR_toolGarra\WObj:=wobjMDF;
        MoveL pDepGaveta_1_91,v1000,z50,USR_toolGarra\WObj:=wobjMDF;
        MoveJ pDepGaveta_1_101,v1000,z50,USR_toolGarra\WObj:=wobjMDF;
    ENDPROC

    PROC mRetiraGaveta_1()
        MoveJ pRetGaveta_1_11,v1000,z50,USR_toolGarra\WObj:=wobjMDF;
        MoveL pRetGaveta_1_1,v1000,z50,USR_toolGarra\WObj:=wobjMDF;
        MoveL pRetGaveta_1_21,v1000,z50,USR_toolGarra\WObj:=wobjMDF;
        !
        ROB_GarraFechar;
        !
        MoveL pRetGaveta_1_31,v1000,z50,USR_toolGarra\WObj:=wobjMDF;
        MoveL pRetGaveta_1_41,v1000,z50,USR_toolGarra\WObj:=wobjMDF;
        MoveL pRetGaveta_1_51,v1000,z50,USR_toolGarra\WObj:=wobjMDF;
        MoveL pRetGaveta_1_61,v1000,z50,USR_toolGarra\WObj:=wobjMDF;
        MoveL pRetGaveta_1_71,v1000,z50,USR_toolGarra\WObj:=wobjMDF;
        MoveL pRetGaveta_1_81,v1000,z50,USR_toolGarra\WObj:=wobjMDF;
        MoveJ pRetGaveta_1_91,v1000,z50,USR_toolGarra\WObj:=wobjMDF;
        MoveJ pRetGaveta_1_101,v1000,z50,USR_toolGarra\WObj:=wobjMDF;
    ENDPROC

    PROC mDepGaveta_2()
        MoveJ pDepGaveta_2_1,v1000,z50,USR_toolGarra\WObj:=wobjMDF;
        MoveJ pDepGaveta_2_11,v1000,z50,USR_toolGarra\WObj:=wobjMDF;
        !
        MoveJ pDepGaveta_2_21,v1000,z50,USR_toolGarra\WObj:=wobjMDF;
        MoveL pDepGaveta_2_31,v1000,z50,USR_toolGarra\WObj:=wobjMDF;
        MoveL pDepGaveta_2_41,v1000,z50,USR_toolGarra\WObj:=wobjMDF;
        MoveL pDepGaveta_2_51,v1000,z50,USR_toolGarra\WObj:=wobjMDF;
        MoveL pDepGaveta_2_61,v1000,z50,USR_toolGarra\WObj:=wobjMDF;
        MoveL pDepGaveta_2_71,v1000,z50,USR_toolGarra\WObj:=wobjMDF;
        !
        ROB_GarraAbrir;
        !
        MoveL pDepGaveta_2_81,v1000,z50,USR_toolGarra\WObj:=wobjMDF;
        MoveL pDepGaveta_2_91,v1000,z50,USR_toolGarra\WObj:=wobjMDF;
        MoveJ pDepGaveta_2_101,v1000,z50,USR_toolGarra\WObj:=wobjMDF;
    ENDPROC

    PROC mRetiraGaveta_2()
        MoveJ pRetGaveta_2_11,v1000,z50,USR_toolGarra\WObj:=wobjMDF;
        MoveL pRetGaveta_2_1,v1000,z50,USR_toolGarra\WObj:=wobjMDF;
        MoveL pRetGaveta_2_21,v1000,z50,USR_toolGarra\WObj:=wobjMDF;
        !
        ROB_GarraFechar;
        !
        MoveL pRetGaveta_2_31,v1000,z50,USR_toolGarra\WObj:=wobjMDF;
        MoveL pRetGaveta_2_41,v1000,z50,USR_toolGarra\WObj:=wobjMDF;
        MoveL pRetGaveta_2_51,v1000,z50,USR_toolGarra\WObj:=wobjMDF;
        MoveL pRetGaveta_2_61,v1000,z50,USR_toolGarra\WObj:=wobjMDF;
        MoveL pRetGaveta_2_71,v1000,z50,USR_toolGarra\WObj:=wobjMDF;
        MoveL pRetGaveta_2_81,v1000,z50,USR_toolGarra\WObj:=wobjMDF;
        MoveJ pRetGaveta_2_91,v1000,z50,USR_toolGarra\WObj:=wobjMDF;
        MoveJ pRetGaveta_2_101,v1000,z50,USR_toolGarra\WObj:=wobjMDF;
    ENDPROC

    PROC mDepGaveta_3()
        MoveJ pDepGaveta_3_1,v1000,z50,USR_toolGarra\WObj:=wobjMDF;
        MoveJ pDepGaveta_3_11,v1000,z50,USR_toolGarra\WObj:=wobjMDF;
        !
        MoveJ pDepGaveta_3_21,v1000,z50,USR_toolGarra\WObj:=wobjMDF;
        MoveL pDepGaveta_3_31,v1000,z50,USR_toolGarra\WObj:=wobjMDF;
        MoveL pDepGaveta_3_41,v1000,z50,USR_toolGarra\WObj:=wobjMDF;
        !MoveL pDepGaveta_3_51,v1000,z50,USR_toolGarra\WObj:=wobjMDF;
        MoveL pDepGaveta_3_61,v1000,z50,USR_toolGarra\WObj:=wobjMDF;
        MoveL pDepGaveta_3_71,v1000,z50,USR_toolGarra\WObj:=wobjMDF;
        MoveL pDepGaveta_3, v1000, fine, USR_toolGarra\WObj:=wobjMDF;
        !
        ROB_GarraAbrir;
        !
        MoveL pDepGaveta_3_81,v1000,z50,USR_toolGarra\WObj:=wobjMDF;
        MoveL pDepGaveta_3_91,v1000,z50,USR_toolGarra\WObj:=wobjMDF;
        MoveJ pDepGaveta_3_101,v1000,z50,USR_toolGarra\WObj:=wobjMDF;
    ENDPROC

    PROC mRetiraGaveta_3()
        MoveJ pRetGaveta_3_11,v1000,z50,USR_toolGarra\WObj:=wobjMDF;
        MoveL pRetGaveta_3_1,v1000,z50,USR_toolGarra\WObj:=wobjMDF;
        MoveL pRetGaveta_3_111, v1000, z50, USR_toolGarra\WObj:=wobjMDF;
        MoveL pRetGaveta_3_21,v1000,z50,USR_toolGarra\WObj:=wobjMDF;
        !
        ROB_GarraFechar;
        !
        MoveL pRetGaveta_3_31,v1000,z50,USR_toolGarra\WObj:=wobjMDF;
        MoveL pRetGaveta_3_41,v1000,z50,USR_toolGarra\WObj:=wobjMDF;
        MoveL pRetGaveta_3_51,v1000,z50,USR_toolGarra\WObj:=wobjMDF;
        MoveL pRetGaveta_3_61,v1000,z50,USR_toolGarra\WObj:=wobjMDF;
        MoveL pRetGaveta_3_71,v1000,z50,USR_toolGarra\WObj:=wobjMDF;
        MoveL pRetGaveta_3_81,v1000,z50,USR_toolGarra\WObj:=wobjMDF;
        MoveJ pRetGaveta_3_91,v1000,z50,USR_toolGarra\WObj:=wobjMDF;
        MoveJ pRetGaveta_3_101,v1000,z50,USR_toolGarra\WObj:=wobjMDF;
    ENDPROC

    PROC mDepGaveta_4()
        MoveJ pDepGaveta_4_1,v1000,z50,USR_toolGarra\WObj:=wobjMDF;
        MoveJ pDepGaveta_4_11,v1000,z50,USR_toolGarra\WObj:=wobjMDF;
        !
        MoveJ pDepGaveta_4_21,v1000,z50,USR_toolGarra\WObj:=wobjMDF;
        MoveL pDepGaveta_4_31,v1000,z50,USR_toolGarra\WObj:=wobjMDF;
        MoveL pDepGaveta_4_41,v1000,z50,USR_toolGarra\WObj:=wobjMDF;
        MoveL pDepGaveta_4_51,v1000,z50,USR_toolGarra\WObj:=wobjMDF;
        MoveL pDepGaveta_4_61,v1000,z50,USR_toolGarra\WObj:=wobjMDF;
        MoveL pDepGaveta_4_71,v1000,z50,USR_toolGarra\WObj:=wobjMDF;
        MoveL pDepGaveta_4,v1000,z50,USR_toolGarra\WObj:=wobjMDF;
        !
        ROB_GarraAbrir;
        !
        MoveL pDepGaveta_4_81,v1000,z50,USR_toolGarra\WObj:=wobjMDF;
        MoveL pDepGaveta_4_111, v1000, z50, USR_toolGarra\WObj:=wobjMDF;
        MoveL pDepGaveta_4_91,v1000,z50,USR_toolGarra\WObj:=wobjMDF;
        MoveJ pDepGaveta_4_101,v1000,z50,USR_toolGarra\WObj:=wobjMDF;
    ENDPROC

    PROC mRetiraGaveta_4()
        MoveJ pRetGaveta_4_11,v1000,z50,USR_toolGarra\WObj:=wobjMDF;
        MoveL pRetGaveta_4_1,v1000,z50,USR_toolGarra\WObj:=wobjMDF;
        MoveL pRetGaveta_4_111, v1000, fine, USR_toolGarra\WObj:=wobjMDF;
        MoveL pRetGaveta_4_21, v1000, fine, USR_toolGarra\WObj:=wobjMDF;
        !
        ROB_GarraFechar;
        !
        MoveL pRetGaveta_4_31,v1000,z50,USR_toolGarra\WObj:=wobjMDF;
        MoveL pRetGaveta_4_41,v1000,z50,USR_toolGarra\WObj:=wobjMDF;
        MoveL pRetGaveta_4_51,v1000,z50,USR_toolGarra\WObj:=wobjMDF;
        MoveL pRetGaveta_4_61,v1000,z50,USR_toolGarra\WObj:=wobjMDF;
        MoveL pRetGaveta_4_71,v1000,z50,USR_toolGarra\WObj:=wobjMDF;
        MoveL pRetGaveta_4_81,v1000,z50,USR_toolGarra\WObj:=wobjMDF;
        MoveJ pRetGaveta_4_91,v1000,z50,USR_toolGarra\WObj:=wobjMDF;
        MoveJ pRetGaveta_4_101,v1000,z50,USR_toolGarra\WObj:=wobjMDF;
    ENDPROC

    PROC mDepGaveta_5()
        MoveJ pDepGaveta_5_1,v1000,z50,USR_toolGarra\WObj:=wobjMDF;
        MoveJ pDepGaveta_5_11,v1000,z50,USR_toolGarra\WObj:=wobjMDF;
        !
        MoveJ pDepGaveta_5_21,v1000,z50,USR_toolGarra\WObj:=wobjMDF;
        MoveL pDepGaveta_5_31,v1000,z50,USR_toolGarra\WObj:=wobjMDF;
        MoveL pDepGaveta_5_41,v1000,z50,USR_toolGarra\WObj:=wobjMDF;
        MoveL pDepGaveta_5_51,v1000,z50,USR_toolGarra\WObj:=wobjMDF;
        MoveL pDepGaveta_5_61,v1000,z50,USR_toolGarra\WObj:=wobjMDF;
        MoveL pDepGaveta_5_71,v1000,z50,USR_toolGarra\WObj:=wobjMDF;
        !
        ROB_GarraAbrir;
        !
        MoveL pDepGaveta_5_81,v1000,z50,USR_toolGarra\WObj:=wobjMDF;
        MoveL pDepGaveta_5_91,v1000,z50,USR_toolGarra\WObj:=wobjMDF;
        MoveJ pDepGaveta_5_101,v1000,z50,USR_toolGarra\WObj:=wobjMDF;
    ENDPROC

    PROC mRetiraGaveta_5()
        MoveJ pRetGaveta_5_11,v1000,z50,USR_toolGarra\WObj:=wobjMDF;
        MoveL pRetGaveta_5_1,v1000,z50,USR_toolGarra\WObj:=wobjMDF;
        MoveL pRetGaveta_5_21,v1000,z50,USR_toolGarra\WObj:=wobjMDF;
        !
        ROB_GarraFechar;
        !
        MoveL pRetGaveta_5_31,v1000,z50,USR_toolGarra\WObj:=wobjMDF;
        MoveL pRetGaveta_5_41,v1000,z50,USR_toolGarra\WObj:=wobjMDF;
        MoveL pRetGaveta_5_51,v1000,z50,USR_toolGarra\WObj:=wobjMDF;
        MoveL pRetGaveta_5_61,v1000,z50,USR_toolGarra\WObj:=wobjMDF;
        MoveL pRetGaveta_5_71,v1000,z50,USR_toolGarra\WObj:=wobjMDF;
        MoveL pRetGaveta_5_81,v1000,z50,USR_toolGarra\WObj:=wobjMDF;
        MoveJ pRetGaveta_5_91,v1000,z50,USR_toolGarra\WObj:=wobjMDF;
        MoveJ pRetGaveta_5_101,v1000,z50,USR_toolGarra\WObj:=wobjMDF;
    ENDPROC

    PROC mDepGaveta_6()
        MoveJ pDepGaveta_6_1,v1000,z50,USR_toolGarra\WObj:=wobjMDF;
        MoveJ pDepGaveta_6_11,v1000,z50,USR_toolGarra\WObj:=wobjMDF;
        !
        MoveJ pDepGaveta_6_21,v1000,z50,USR_toolGarra\WObj:=wobjMDF;
        MoveL pDepGaveta_6_31,v1000,z50,USR_toolGarra\WObj:=wobjMDF;
        MoveL pDepGaveta_6_41,v1000,z50,USR_toolGarra\WObj:=wobjMDF;
        MoveL pDepGaveta_6_51,v1000,z50,USR_toolGarra\WObj:=wobjMDF;
        MoveL pDepGaveta_6_61,v1000,z50,USR_toolGarra\WObj:=wobjMDF;
        MoveL pDepGaveta_6_71,v1000,z50,USR_toolGarra\WObj:=wobjMDF;
        !
        ROB_GarraAbrir;
        !
        MoveL pDepGaveta_6_81,v1000,z50,USR_toolGarra\WObj:=wobjMDF;
        MoveL pDepGaveta_6_91,v1000,z50,USR_toolGarra\WObj:=wobjMDF;
        MoveJ pDepGaveta_6_101,v1000,z50,USR_toolGarra\WObj:=wobjMDF;
    ENDPROC

    PROC mRetiraGaveta_6()
        MoveJ pRetGaveta_6_11,v1000,z50,USR_toolGarra\WObj:=wobjMDF;
        MoveL pRetGaveta_6_1,v1000,z50,USR_toolGarra\WObj:=wobjMDF;
        MoveL pRetGaveta_6_21,v1000,z50,USR_toolGarra\WObj:=wobjMDF;
        !
        ROB_GarraFechar;
        !
        MoveL pRetGaveta_6_31,v1000,z50,USR_toolGarra\WObj:=wobjMDF;
        MoveL pRetGaveta_6_41,v1000,z50,USR_toolGarra\WObj:=wobjMDF;
        MoveL pRetGaveta_6_51,v1000,z50,USR_toolGarra\WObj:=wobjMDF;
        MoveL pRetGaveta_6_61,v1000,z50,USR_toolGarra\WObj:=wobjMDF;
        MoveL pRetGaveta_6_71,v1000,z50,USR_toolGarra\WObj:=wobjMDF;
        MoveL pRetGaveta_6_81,v1000,z50,USR_toolGarra\WObj:=wobjMDF;
        MoveJ pRetGaveta_6_91,v1000,z50,USR_toolGarra\WObj:=wobjMDF;
        MoveJ pRetGaveta_6_101,v1000,z50,USR_toolGarra\WObj:=wobjMDF;
    ENDPROC

ENDMODULE
